(*

.. <legal notes>

legal notes
=================
| SPDX-FileCopyrightText: © 2025 Oleksandr Tiutyk <trofimich@gmail.com>
| SPDX-License-Identifier: LGPL-3.0-only
| For details check: LGPL-3.0-only_

.. _LGPL-3.0-only: https://www.gnu.org/licenses/lgpl-3.0.en.html

.. </legal notes>

*)

INTERFACE ITask EXTENDS TOF_Core.IExecutable

{attribute 'monitoring' := 'call'}
PROPERTY AbortReason : REFERENCE TO WSTRING(255)
GET
END_GET
END_PROPERTY

{attribute 'monitoring' := 'call'}
PROPERTY ErrorMessage : REFERENCE TO ERROR_MESSAGE
GET
END_GET
END_PROPERTY

{attribute 'monitoring' := 'call'}
PROPERTY InTransition : BOOL
GET
END_GET
END_PROPERTY

{attribute 'monitoring' := 'call'}
PROPERTY Name : WSTRING
GET
END_GET
SET
END_SET
END_PROPERTY

METHOD RequestCancel : BOOL
VAR_OUTPUT
	refuseReason : WSTRING(255);
END_VAR
END_METHOD

METHOD RequestStart : BOOL
VAR_OUTPUT
	refuseReason : WSTRING(255);
END_VAR
END_METHOD

METHOD Reset : BOOL
VAR_OUTPUT
	refuseReason : WSTRING(255);
END_VAR
END_METHOD

{attribute 'monitoring' := 'call'}
PROPERTY State : TASK_STATE
GET
END_GET
END_PROPERTY

{attribute 'monitoring' := 'call'}
PROPERTY StateChanged : BOOL
GET
END_GET
END_PROPERTY

END_INTERFACE

(* stored: Version 1.1.0.1
   Itf ITask: Id {575cbb28-8594-44fa-869a-33267f7f0a3c}
   Property AbortReason: Id {3bee27f3-ca68-4599-807e-089fd46d8985}
   Get Get: Id {ec839d45-850d-4c19-b67a-5fc1dcc5f6f0}
   Property ErrorMessage: Id {693d2592-f5a7-4888-b697-1ffc6dc94875}
   Get Get: Id {6e4e51d2-2b44-434d-ac43-b5b87e18a0e6}
   Property InTransition: Id {e518ed3b-ec73-44f5-82d8-95864b918b31}
   Get Get: Id {a496d9a0-4868-494b-9cf1-c26df5e59eee}
   Property Name: Id {2ef62023-cb7d-409a-b3ca-14708401cfe3}
   Get Get: Id {53ffbb66-56d7-495a-b74d-0266b759f46f}
   Set Set: Id {6e96319c-2ab1-4bbe-a76a-9f15d9024330}
   Method RequestCancel: Id {21c2e6f7-d1a2-4506-8e1a-380eaea2af15}
   Method RequestStart: Id {023400b1-c0d4-4a01-bff1-7b11703d2edd}
   Method Reset: Id {5660a6b5-d1d8-4613-b3d7-6b389efa0396}
   Property State: Id {26c74757-65ff-4b56-905a-dd3b6818504d}
   Get Get: Id {ed4dc31d-6997-4ba2-a9fc-5072257adf60}
   Property StateChanged: Id {3ed7e09a-556a-4fde-ac03-7e897c90bd36}
   Get Get: Id {12361e09-ab1c-49ab-9369-c864183e37be} *)
